(* CODESYS project CtaAppHysterese_1.0.0.0.library
   Description: Hysterese Library der CTA
   Version: 1.0.0.0
   Title: CtaAppHysterese
   Author: SIS
   LanguageModelAttribute: qualified-access-only
   DocFormat: reStructuredText
   Placeholder: CtaAppHysterese
   DefaultNamespace: CtaAppHysterese
   CompiledLibraryCompatibilityVersion: CODESYS V3.5 SP16 Patch 3
   Company: CTA

Project tree, tasks and I/O mapping:
  libraries: VisuSymbols, 4.5.0.0 (System)
  40 Visualizations/
  30 Program Organization Units/
    function block fbHyst_Dir [ST]
    function block fbHyst_Rev [ST]
  00000000-0000-0000-0000-000000000000|D:\CoDeSys\LibrariesV3\trunk\Intern\CAA\CAA Template\3.4.0.0 draft\Placeholder.xml
  00000000-0000-0000-0000-000000000000|D:\CoDeSys\LibrariesV3\trunk\Intern\CAA\CAA Template\3.2.0.3 draft\Prefix.pdf
  00000000-0000-0000-0000-000000000000|D:\CoDeSys\LibrariesV3\trunk\Intern\CAA\CAA Template\3.5.2.0 draft\Placeholder.xml
  20 Structs/
  50 Images/
  10 Documenation/
    global variables VersionHistory
    global variables readMe
  21 Interface/
  11 Library Parameter/
  12 Konstanten/
  60 Textlisten/
  13 Globale Variablen/
*)

// 10 Documenation/VersionHistory
(* 

.. image:: ../../Images/CTA_Logo.jpg
   :align: right
   :width: 15% 

**Vorlage**   


============ =========== =========== ============================================
**Date**     **Version** **Author**  **Change**
------------ ----------- ----------- --------------------------------------------
04.03.2021   0.0.0.0     SIS         Vorlage erstellt

============ =========== =========== ============================================


*)
VAR_GLOBAL
    stInfo : STRING:= '0.0.0.0, Vorlage, CTA';
END_VAR

// 10 Documenation/readMe
(*

**ReadMe**
 
|	**Empfehlung**
|
|	Dokumentrieren Sie die Library für eine nachhaltige Entwicklung
|     
| *Beispiel* 
|
| Dies ist die Vorlage Library der CTA. Erstellen Sie ihre Library anhand dieser Vorlage.
*)

VAR_GLOBAL
    xReadMeDone              :   BOOL;
END_VAR

// 30 Program Organization Units/fbHyst_Dir
FUNCTION_BLOCK fbHyst_Dir 
VAR_INPUT
    rIn         :   REAL;
    rSet        :   REAL;
    rDiffOn     :   REAL;
    rDIffOff    :   REAL;
END_VAR
VAR_OUTPUT
    xOut        :   BOOL;
END_VAR
VAR
END_VAR

IF rIn >= rSet + rDiffOn THEN
    xOut := TRUE;
ELSIF rIn <= rSet - rDIffOff THEN
    xOut := FALSE;
END_IF;

END_FUNCTION_BLOCK

// 30 Program Organization Units/fbHyst_Rev
FUNCTION_BLOCK  fbHyst_Rev 
VAR_INPUT
    rIn         :   REAL;
    rSet        :   REAL;
    rDiffOn     :   REAL;
    rDIffOff    :   REAL;
END_VAR
VAR_OUTPUT
    xOut        :   BOOL;
END_VAR
VAR
    fbHyst_Dir : fbHyst_Dir;
END_VAR

fbHyst_Dir( rIn         :=  rIn,
            rSet        := rSet,
            rDiffOn     := rDIffOff,
            rDIffOff    := rDiffOn,
            xOut        => xOut);

xOut := NOT xOut;

END_FUNCTION_BLOCK
